PROGRAM Fault_Logic
VAR
	
	ScrapBinFullWarning: BOOL;
	RibHopperEmptyFault: BOOL;
	RibHopperNearEmptyWarning: BOOL;
	RibMeasureFault: BOOL;
	LowAirPresFault: BOOL;
	GuardOpenFault: BOOL;
	MotorFault: BOOL;
	JamFault: BOOL;
	AirPresTon : TON;
	AirPresElapsed: TIME;
	
	
	
END_VAR

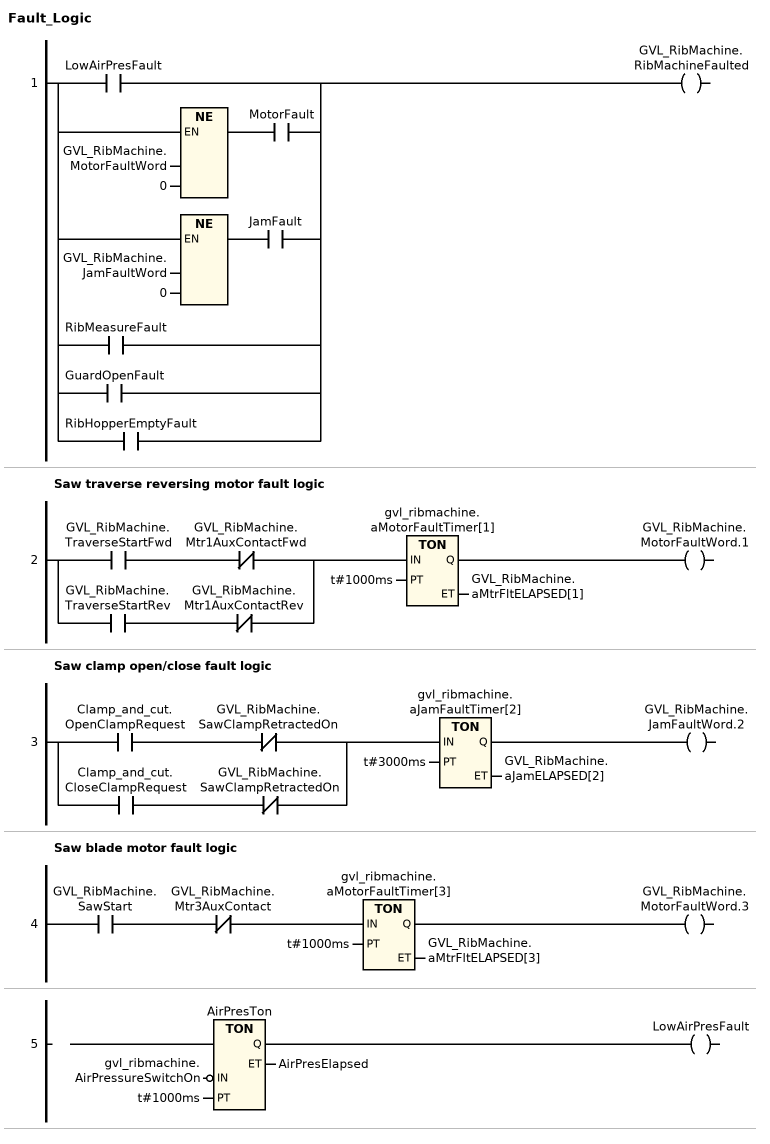
// NETWORK 1
GVL_RibMachine.RibMachineFaulted := LowAirPresFault OR GVL_RibMachine.MotorFaultWord <> 0 AND MotorFault OR GVL_RibMachine.JamFaultWord <> 0 AND JamFault OR RibMeasureFault OR GuardOpenFault OR RibHopperEmptyFault;

// NETWORK 2: Saw traverse reversing motor fault logic
gvl_ribmachine.aMotorFaultTimer[1](
    IN := GVL_RibMachine.TraverseStartFwd AND NOT GVL_RibMachine.Mtr1AuxContactFwd OR GVL_RibMachine.TraverseStartRev AND NOT GVL_RibMachine.Mtr1AuxContactRev,
    PT := t#1000ms,
    ET => GVL_RibMachine.aMtrFltELAPSED[1]); // TON
GVL_RibMachine.MotorFaultWord.1 := gvl_ribmachine.aMotorFaultTimer[1].Q;

// NETWORK 3: Saw clamp open/close fault logic
gvl_ribmachine.aJamFaultTimer[2](
    IN := Clamp_and_cut.OpenClampRequest AND NOT GVL_RibMachine.SawClampRetractedOn OR Clamp_and_cut.CloseClampRequest AND NOT GVL_RibMachine.SawClampRetractedOn,
    PT := t#3000ms,
    ET => GVL_RibMachine.aJamELAPSED[2]); // TON
GVL_RibMachine.JamFaultWord.2 := gvl_ribmachine.aJamFaultTimer[2].Q;

// NETWORK 4: Saw blade motor fault logic
gvl_ribmachine.aMotorFaultTimer[3](
    IN := GVL_RibMachine.SawStart AND NOT GVL_RibMachine.Mtr3AuxContact,
    PT := t#1000ms,
    ET => GVL_RibMachine.aMtrFltELAPSED[3]); // TON
GVL_RibMachine.MotorFaultWord.3 := gvl_ribmachine.aMotorFaultTimer[3].Q;

// NETWORK 5
AirPresTon(IN := NOT gvl_ribmachine.AirPressureSwitchOn, PT := t#1000ms, ET => AirPresElapsed); // TON
LowAirPresFault := AirPresTon.Q;

END_PROGRAM

(* stored: Version 1.1.0.1, ProductVersion 3.1.4024.12
   POU Fault_Logic: Id {30023c80-180b-4024-bf6d-e2b08e247a31}, SpecialFunc None *)
